// TIA Portal project "Lab7" (V16)

(* hardware
DEVICE "S71500/ET200MP station_1"  S7-1500 station
   slot 0: "Rail_0"  Rack  6ES7 590-1***0-0AA0
   slot 1: "PLC_1"  CPU 1512C-1 PN  6ES7 512-1CK00-0AB0  V2.8
      slot 3: "CPU display_1"  6ES7591-1AA00-0AA0
      slot 32768: "PROFINET interface_1"  X1
         slot 32769: "Port_1"  X1 P1
         slot 32770: "Port_2"  X1 P2
      slot 34817: "Virtual CP interface port_1"  Virtual CP interface port  Virtual CP interface port
*)

// ===== PLC "PLC_1"  CPU 1512C-1 PN =====

DATA_BLOCK "PROC_C_DB"   // DB50
{ S7_Optimized_Access := 'TRUE' }
AUTHOR : HHM
FAMILY : PROC_SIM
NAME : PROC_C
VERSION : 1.0
// stored: InstanceOfName PROC_C
"PROC_C"
BEGIN
END_DATA_BLOCK

DATA_BLOCK "MyPID_DB"   // DB200
{ S7_Optimized_Access := 'TRUE' }
AUTHOR : HHManh
FAMILY : AT74_07
NAME : MyPID
VERSION : 1.0
// stored: InstanceOfName MyPID
"MyPID"
BEGIN
END_DATA_BLOCK

FUNCTION_BLOCK "PROC_C"   // FB50, SCL
TITLE = 'process simulation for continious PID controller'
{ S7_Optimized_Access := 'TRUE' }
AUTHOR : HHM
FAMILY : PROC_SIM
NAME : PROC_C
VERSION : 1.0
// KNOW_HOW_PROTECT
   VAR_INPUT
      INV : Real;   // input variable
      DISV : Real;   // disturbance variable
      GAIN : Real := 1.0;   // proportional gain
      TM_LAG1 : Time := T#10S;   // time lag 1
      TM_LAG2 : Time := T#10S;   // time lag 2
      TM_LAG3 : Time := T#10S;   // time lag 3
      COM_RST : Bool;   // complete restart
      CYCLE : Time := T#1S;   // sample time
   END_VAR
   VAR_OUTPUT
      OUTV : Real;   // output variable
   END_VAR
   VAR
      sRueck1 : Real;   // feedback path value 1
      sRueck2 : Real;   // feedback path value 2
      sRueck3 : Real;   // feedback path value 3
   END_VAR
   VAR_TEMP
      Hvar : Real;   // help variable
      rCycle : Real;   // cycle to real
      rTmLag1 : Real;   // time lag 1 to real
      rTmLag2 : Real;   // time lag 2 to real
      rTmLag3 : Real;   // time lag 3 to real
      OutvNew : Real;   // new output variable
   END_VAR
BEGIN
       IF #COM_RST THEN
           #OUTV := #INV;
           #sRueck1 := #OUTV;
           #sRueck2 := #OUTV;
           #sRueck3 := #OUTV;
       ELSE
           #rCycle := DINT_TO_REAL(TIME_TO_DINT(#CYCLE));
           #rTmLag1 := DINT_TO_REAL(TIME_TO_DINT(#TM_LAG1));
           #rTmLag2 := DINT_TO_REAL(TIME_TO_DINT(#TM_LAG2));
           #rTmLag3 := DINT_TO_REAL(TIME_TO_DINT(#TM_LAG3));

           IF #rTmLag1 < #rCycle * 0.5 THEN
               #rTmLag1 := #rCycle * 0.5;
           END_IF;
           IF #rTmLag2 < #rCycle * 0.5 THEN
               #rTmLag2 := #rCycle * 0.5;
           END_IF;
           IF #rTmLag3 < #rCycle * 0.5 THEN
               #rTmLag3 := #rCycle * 0.5;
           END_IF;

           #Hvar := #rCycle / (2.0 * #rTmLag1);
           #Hvar := ((#INV + #DISV) * #GAIN - #sRueck1) * #Hvar / (1.0 + #Hvar);
           #OutvNew := #sRueck1 + #Hvar;
           #sRueck1 := #sRueck1 + 2.0 * #Hvar;

           #Hvar := #rCycle / (2.0 * #rTmLag2);
           #Hvar := (#OutvNew - #sRueck2) * #Hvar / (1.0 + #Hvar);
           #OutvNew := #sRueck2 + #Hvar;
           #sRueck2 := #sRueck2 + 2.0 * #Hvar;

           #Hvar := #rCycle / (2.0 * #rTmLag3);
           #Hvar := (#OutvNew - #sRueck3) * #Hvar / (1.0 + #Hvar);
           #OutvNew := #sRueck3 + #Hvar;
           #sRueck3 := #sRueck3 + 2.0 * #Hvar;

           #OUTV := #OutvNew;
       END_IF;
END_FUNCTION_BLOCK

FUNCTION_BLOCK "MyPID"   // FB200, SCL
TITLE = 'PID-algorithm'
{ S7_Optimized_Access := 'TRUE' }
AUTHOR : HHManh
FAMILY : AT74_07
NAME : MyPID
VERSION : 1.0
// KNOW_HOW_PROTECT
// ---------------------------------------------------------------------------------------
// VARIABLES INPUT DECLARATION
// ---------------------------------------------------------------------------------------
   VAR_INPUT
      COM_RST : Bool := FALSE;   // Complete restart
      CO_TYPE : Bool := FALSE;   // Controller TYPE: 1=direct; 0=reverse
      MAN_ON : Bool := TRUE;   // Manual mode enable
      P_SEL : Bool := TRUE;   // Selecting proportional component
      I_SEL : Bool := TRUE;   // Selecting integral component
      D_SEL : Bool := FALSE;   // Selecting differential component
      SPT_SEL : Bool := TRUE;   // Selecting setpoint tracking
      CYCLE : Time := T#100MS;   // Execution cycle time
      PV : Real;   // Process variable input (%)
      KC : Real := 1.0;   // The proportional gain
      TI : Time := T#20S;   // Integration time
      TD : Time := T#10S;   // Differentiation time
      CO_HLM : Real := 100.0;   // Upper limit of output
      CO_LLM : Real := 0.0;   // Lower limit of output---------------------------------------------------------------------------------------VARIABLES OUTPUT DECLARATION---------------------------------------------------------------------------------------
   END_VAR
   VAR_OUTPUT
      CO : Real;   // Controller output (%)
      QCO_HLM : Bool;   // Upper limit of output reached
      QCO_LLM : Bool;   // Lower limit of output reached
      LMN_P : Real;   // Proportional component
      LMN_I : Real;   // Integral component
      LMN_D : Real;   // Differential component
      PV_OUT : Real;   // Process variable
      ER : Real;   // Error signal---------------------------------------------------------------------------------------VARIABLES INPUT/OUTPUT DECLARATION---------------------------------------------------------------------------------------
   END_VAR
   VAR_IN_OUT
      SP : Real;   // Setpoint (%)
      MAN : Real;   // Manual value for output (%)---------------------------------------------------------------------------------------STATIC VARIABLES INPUT DECLARATION---------------------------------------------------------------------------------------
   END_VAR
   VAR
      LmnI : Real := 0.0;   // I portion
      BIAS : Real := 0.0;   // BIAS value
      lastLmnP : Real := 0.0;   // Last value of P portion
      sCOHLmOn : Bool := FALSE;   // Static variable: output reached high limit
      sCOLLmOn : Bool := FALSE;   // Static variable: output reached low limit---------------------------------------------------------------------------------------TEMPORATY VARIABLES INPUT DECLARATION---------------------------------------------------------------------------------------
   END_VAR
   VAR_TEMP
      CO_temp : Real;   // Temporary variable for controller output
      LmnD : Real;   // D portion
      LmnP : Real;   // P portion
      rCycle : Real;   // Cycle time in REAL
      rTi : Real;   // Integration time in REAL
      rTd : Real;   // Differential time in REAL
      integralDiff : Real;   // Differece in Integral---------------------------------------------------------------------------------------CODE BEGINS---------------------------------------------------------------------------------------
   END_VAR
BEGIN

   IF #COM_RST THEN //If complete restart is activated
       //---------------------------------------------------------------------------------------
       //RESET
       //---------------------------------------------------------------------------------------
       #BIAS := 0.0;
       #LmnP := 0.0;
       #LmnI := 0.0;
       #LmnD := 0.0;
       #lastLmnP := 0.0;
       #CO := 0.0; //Output value
       #QCO_HLM := 0; //Reset upper limit of output achieved bit
       #QCO_LLM := 0; //Reset lower limit of output achieved bit
       #LMN_P := 0.0; //Reset the output of proportional component
       #LMN_I := 0.0; //Reset the output of integral component
       #LMN_D := 0.0; //Reset the output of differential component
       #PV_OUT := 0.0;//Reset the output of process value
       #SP := 0.0; //Reset setpoint
       #MAN := 0.0; //Reset the manual value
       #ER := 0.0; //Reset error
       #sCOHLmOn := FALSE; //Reset the internal var high limit for ouput
       #sCOLLmOn := FALSE; //Reset the internal var low limit for output
   ELSE
       //---------------------------------------------------------------------------------------
       //CONVERSION TO REAL NUMBERS
       //---------------------------------------------------------------------------------------
       #rCycle := DINT_TO_REAL(TIME_TO_DINT(#CYCLE)) / 1000.0; //CYCLE->secs & real
       #rTi := DINT_TO_REAL(TIME_TO_DINT(#TI)) / 1000.0;//TI->sec&Real
       #rTd := DINT_TO_REAL(TIME_TO_DINT(#TD)) / 1000.0;//TD->secs&Real
       //---------------------------------------------------------------------------------------
       //CHECKING TYPE: REVERSE or DIRECT
       //The controller is REVERSE if TYPE=0; and DIRECT if TYPE=1.The method to calculate the
       // error depending on the TYPE.
       //---------------------------------------------------------------------------------------
       IF (NOT #CO_TYPE) THEN
           #ER := #SP - #PV;
       ELSE
           #ER := #PV - #SP;
       END_IF;

       //THE PROPORTIONAL COMPONENT: This is always calculated but may contribute to the 
       //controller output or displayed if the proportional mode is selected.
       #LmnP := #KC * #ER;
       //---------------------------------------------------------------------------------------
       //CONTROLER IN MANUAL MODE
       //---------------------------------------------------------------------------------------
       IF #MAN_ON THEN
           #BIAS := #MAN;
           #CO_temp := #BIAS; //Output value will be MAN
           //The integration is back-calculated at MAN mode so that a bumpless transfer is 
           //archieved when switching to AUTO mode (there won't be an aprupt change in 
           //controller output).
           #LmnI := #CO_temp - #LmnP - #BIAS;
           #LmnD := 0.0;
           //In case integration isn't slected for auto mode, then setpoint tracking 
           //should be selected to get the bumpless transfer.
           IF #SPT_SEL THEN
               #SP := #PV;
           END_IF;
           //--------------------------------------------------------------------------------------
           //CONTROLLER IN AUTO MODE
           //--------------------------------------------------------------------------------------
       ELSE
           //The integral portion is computed only if the integral mode is selected
           //otherwise it is reset to 0.0%
           IF #I_SEL THEN
               //If the integral difference is positive and the CO has reached highlimit or if
               //it is negative and the CO has reached low limit, the integral difference
               //is reset to 0.0% so that the integral portion is kept unchanged.
               IF ((#integralDiff > 0.0) AND #sCOHLmOn) OR ((#integralDiff < 0.0) AND #sCOLLmOn)
               THEN
                   #integralDiff := 0.0;
               ELSE
                   #integralDiff := (#rCycle / #rTi) * #LmnP;
               END_IF;
               #LmnI := #LmnI + #integralDiff;
               //Windup reset
               //If integral portion and controller output are over the limit, the integration will
               //be adjusted to keep the controller output at limits.
               IF (#LmnI > #CO_HLM) AND (#CO_temp > #CO_HLM) THEN
                   #LmnI := #LmnI - (#CO_temp - #CO_HLM);
               ELSIF (#LmnI < #CO_LLM) AND (#CO_temp < #CO_LLM) THEN
                   #LmnI := #LmnI + (#CO_HLM - #CO_temp);
               END_IF;

           ELSE
               #LmnI := 0.0;
           END_IF;
           //The derivative is computed only in auto and derivative mode is selected otherwise
           // it is reset TO 0.0%
           IF #D_SEL THEN
               #LmnD := (#rTd / #rCycle) * (#LmnP - #lastLmnP);
               #lastLmnP := #LmnP;
           ELSE
               #LmnD := 0.0;
           END_IF;
           //If proportional mode is slected then proportional portion will be contributed to
           //the output controller otherwise not.   
           IF #P_SEL THEN
               #CO_temp := #BIAS + #LmnP + #LmnI + #LmnD;
           ELSE
               #CO_temp := #BIAS + #LmnI + #LmnD;
           END_IF;
           //To get a  bumpless transfer when switching to MAN mode, the manual value (MAN)
           //must be adjusted to the current value of the controller ouput.
           #MAN := #CO_temp;

       END_IF;
       //--------------------------------------------------------------------------------------
       //LIMIT LOGIC: If the controller output is over the limits,it is kept at limits and
       // digital alarms are set.
       //--------------------------------------------------------------------------------------
       #sCOHLmOn := 0;
       #sCOLLmOn := 0;
       IF (#CO_temp >= #CO_HLM)
       THEN
           #QCO_HLM := 1;
           #QCO_LLM := 0;
           #CO_temp := #CO_HLM;
           #sCOHLmOn := 1;
       ELSE
           #QCO_HLM := 0;
           IF (#CO_temp <= #CO_LLM)
           THEN
               #QCO_LLM := 1;
               #CO_temp := #CO_LLM;
               #sCOLLmOn := 1;
           ELSE
               #QCO_LLM := 0;
           END_IF;
       END_IF;
       //--------------------------------------------------------------------------------------
       //OUTPUTING VALUES
       //--------------------------------------------------------------------------------------
       #PV_OUT := #PV; //Displaying process variable
       #LMN_P := #LmnP; //Displaying propotional portion
       #LMN_I := #LmnI; //Displaying integral portion
       #LMN_D := #LmnD; //Displaying derivative portion
       #CO := #CO_temp; //Sending the value to controller output

   END_IF;
END_FUNCTION_BLOCK

ORGANIZATION_BLOCK "Main"   // OB1, LAD, ProgramCycle
TITLE = "Main Program Sweep (Cycle)"
{ S7_Optimized_Access := 'TRUE' }
VERSION : 0.1
   VAR_INPUT
      Initial_Call : Bool;   // Initial call of this OB
      Remanence : Bool;   // =True, if remanent data are available
   END_VAR
   VAR_TEMP   // added for the SCL form of the ladder/FBD networks
      _w1 : Bool;
   END_VAR
BEGIN

REGION Network 1
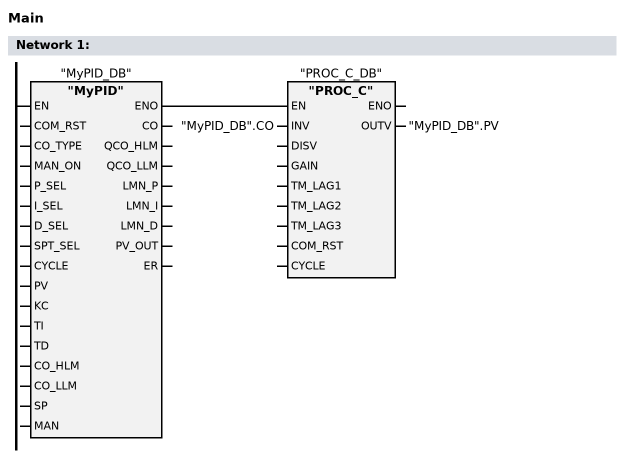
   RUNG wire#powerrail
      "MyPID_DB"(COM_RST :=, CO_TYPE :=, MAN_ON :=, P_SEL :=, I_SEL :=, D_SEL :=, SPT_SEL :=, CYCLE :=, PV :=, KC :=, TI :=, TD :=, CO_HLM :=, CO_LLM :=, SP :=, MAN :=, CO =>, QCO_HLM =>, QCO_LLM =>, LMN_P =>, LMN_I =>, LMN_D =>, PV_OUT =>, ER =>)
      "PROC_C_DB"(INV := "MyPID_DB".CO, DISV :=, GAIN :=, TM_LAG1 :=, TM_LAG2 :=, TM_LAG3 :=, COM_RST :=, CYCLE :=, OUTV => "MyPID_DB".PV)
   END_RUNG
   // the same network as SCL:
   "MyPID_DB"(ENO => #_w1);   // "MyPID"
   IF #_w1 THEN
       "PROC_C_DB"(INV := "MyPID_DB".CO, OUTV => "MyPID_DB".PV);   // "PROC_C"
   END_IF;
END_REGION
END_ORGANIZATION_BLOCK

ORGANIZATION_BLOCK "Cyclic interrupt"   // OB35, LAD, CyclicInterrupt
{ S7_Optimized_Access := 'TRUE' }
VERSION : 0.1
   VAR_INPUT
      Initial_Call : Bool;   // Initial call of this OB
      Event_Count : Int;   // Events discarded
   END_VAR
BEGIN
END_ORGANIZATION_BLOCK